{attribute 'linkalways'}
{attribute 'no_explicit_call' := 'This FB is a CLASS and must be accessed using methods or properties'}
FUNCTION_BLOCK DefaultFileLogEventFormatter IMPLEMENTS LogEventFormatter
VAR
END_VAR

METHOD PUBLIC Format : T_MaxString
VAR_INPUT
	event : LogEvent;
END_VAR
VAR_INST
	{attribute 'hide'}
	message_builder : StringBuilder;
END_VAR
VAR CONSTANT
	DELIMITER : STRING := '|';
END_VAR
Format := message_builder
	.Reset()
	.Append(Tc2_Utilities.SystemTime_To_String(event.timestamp))
	.Append(DELIMITER)
	.Append(TO_STRING(event.level))
	.Append(DELIMITER)
	.Append(event.logger)
	.Append(DELIMITER)
	.Append(event.message)
	.ToString();
END_METHOD

END_FUNCTION_BLOCK

(* stored: Version 1.1.0.1
   POU DefaultFileLogEventFormatter: Id {aa68e43a-1202-4457-87ae-37bbd3c75af4}, SpecialFunc None
   Method Format: Id {79736781-e417-4725-b09d-6898db45937f} *)
